TYPE stHMIMotorisedCB :
STRUCT
END_STRUCT
END_TYPE

(* stored: Version 1.1.0.1, ProductVersion 3.1.4024.11
   DUT stHMIMotorisedCB: Id {a4c8b693-efa3-426d-8c95-d3cb6ef3ad2b} *)
